PROGRAM Stn051_PrgCalls
VAR
END_VAR

//Turn on the default programs
IF gFirstScan THEN
	gDebug_ComponentCall.CallStn051_20_ReturnBreakStopsGrn := TRUE;
	gDebug_ComponentCall.CallStn051_21_ReturnBreakStopsRed := TRUE;
END_IF

IF gDebug_ComponentCall.CallStn051_20_ReturnBreakStopsGrn OR
		gFirstScan THEN
	Stn051_20_ReturnBreakStopsGrn();
END_IF

IF gDebug_ComponentCall.CallStn051_21_ReturnBreakStopsRed OR
		gFirstScan THEN
	Stn051_21_ReturnBreakStopsRed();
END_IF

END_PROGRAM

(* stored: Version 1.1.0.1, ProductVersion 3.1.4024.6
   POU Stn051_PrgCalls: Id {7c356480-98ab-4cc5-9a93-1cd8a1ba97df}, SpecialFunc None *)
